// SIMATIC S7-200 project (STEP 7-Micro/WIN), CPU 224XP REL 02.01

SYMBOL_TABLE USUARIO1
S_LENTO          I0.0
S_RAPIDO         I0.1
B_LENTO          I0.2
B_RAPIDO         I0.3
D_LENTO          I0.4
D_RAPIDO         I0.5
I_LENTO          I0.6
I_RAPIDO         I0.7
FC_BAJADA        I1.0
FC_SUBIDA        I1.1
FC_IZQUIERDA     I1.2
FC_DERECHA       I1.3
M1_S_U1V1W1TSR   Q0.0
M1_S_U2V2W2_TSR  Q0.1
M1_SB_CORTOCIRQUITADO Q0.2
M1_B_U1V1W1_RST  Q0.3
M1_B_U2V2W2_RST  Q0.4
M2_D_U1V1W1_RST  Q0.5
M2_D_U2V2W2_RST  Q0.6
M2_DI_CORTOCIRQUITADO Q0.7
M2_I_U1V1W1_TSR  Q1.0
M2_I_U2V2W2_TSR  Q1.1
END_SYMBOL_TABLE

ORGANIZATION_BLOCK PRINCIPAL:OB1
TITLE=COMENTARIOS DEL PROGRAMA
BEGIN
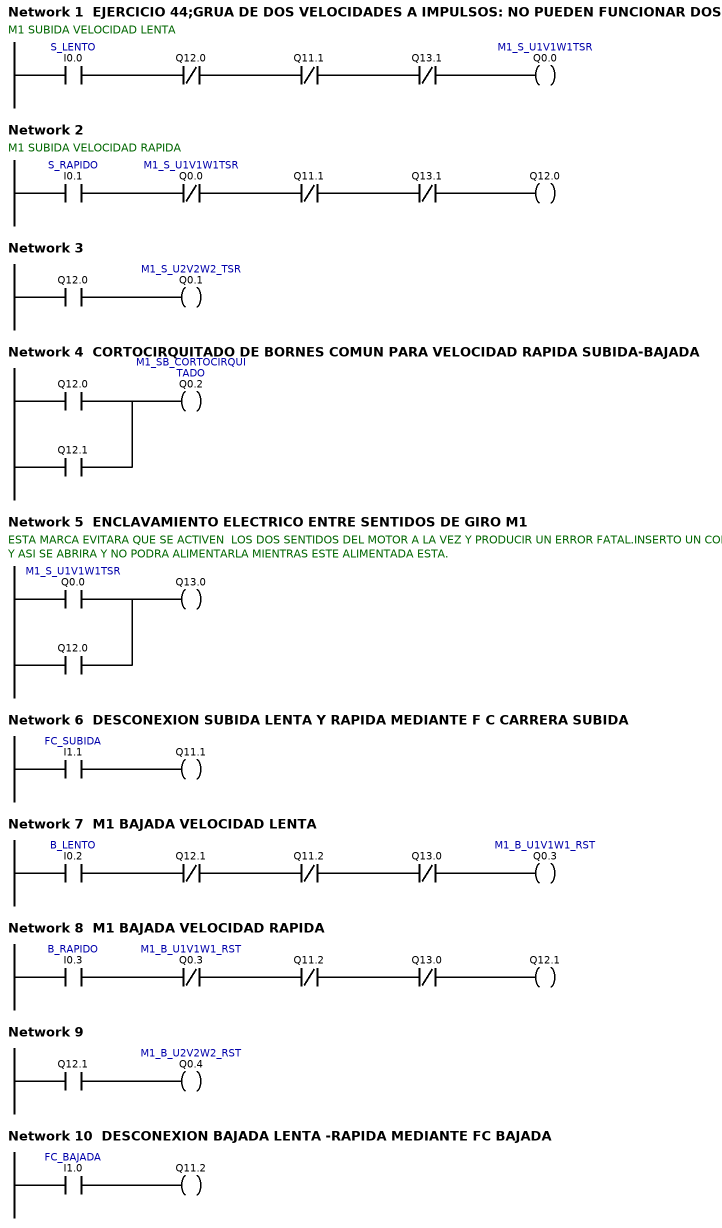
Network 1 // EJERCICIO 44;GRUA DE DOS VELOCIDADES A IMPULSOS:
NO PUEDEN FUNCIONAR DOS VELOCIDADES DEL MISMO SENTIDO A LA VEZ Y TAMPOCO DOS SENTIDOS DEL MISMO MOTOR.
// M1 SUBIDA VELOCIDAD LENTA
LD     S_LENTO:I0.0
AN     Q12.0
AN     Q11.1
AN     Q13.1
=      M1_S_U1V1W1TSR:Q0.0
Network 2
// M1 SUBIDA VELOCIDAD RAPIDA
LD     S_RAPIDO:I0.1
AN     M1_S_U1V1W1TSR:Q0.0
AN     Q11.1
AN     Q13.1
=      Q12.0
Network 3
LD     Q12.0
=      M1_S_U2V2W2_TSR:Q0.1
Network 4 // CORTOCIRQUITADO DE BORNES COMUN PARA VELOCIDAD RAPIDA SUBIDA-BAJADA
LD     Q12.0
O      Q12.1
=      M1_SB_CORTOCIRQUITADO:Q0.2
Network 5 // ENCLAVAMIENTO ELECTRICO ENTRE SENTIDOS DE GIRO M1
// ESTA MARCA EVITARA QUE SE ACTIVEN  LOS DOS SENTIDOS DEL MOTOR A LA VEZ Y PRODUCIR UN ERROR FATAL.INSERTO UN CONTACTO CERRADO DELANTE DE LA BOBINA DEL SENTIDO CONTRARIO Y ASI SE ABRIRA Y NO PODRA ALIMENTARLA MIENTRAS ESTE ALIMENTADA ESTA.
LD     M1_S_U1V1W1TSR:Q0.0
O      Q12.0
=      Q13.0
Network 6 // DESCONEXION SUBIDA LENTA Y RAPIDA MEDIANTE F C CARRERA SUBIDA
LD     FC_SUBIDA:I1.1
=      Q11.1
Network 7 // M1 BAJADA VELOCIDAD LENTA 
LD     B_LENTO:I0.2
AN     Q12.1
AN     Q11.2
AN     Q13.0
=      M1_B_U1V1W1_RST:Q0.3
Network 8 // M1 BAJADA VELOCIDAD RAPIDA
LD     B_RAPIDO:I0.3
AN     M1_B_U1V1W1_RST:Q0.3
AN     Q11.2
AN     Q13.0
=      Q12.1
Network 9
LD     Q12.1
=      M1_B_U2V2W2_RST:Q0.4
Network 10 // DESCONEXION BAJADA LENTA -RAPIDA MEDIANTE FC BAJADA
LD     FC_BAJADA:I1.0
=      Q11.2
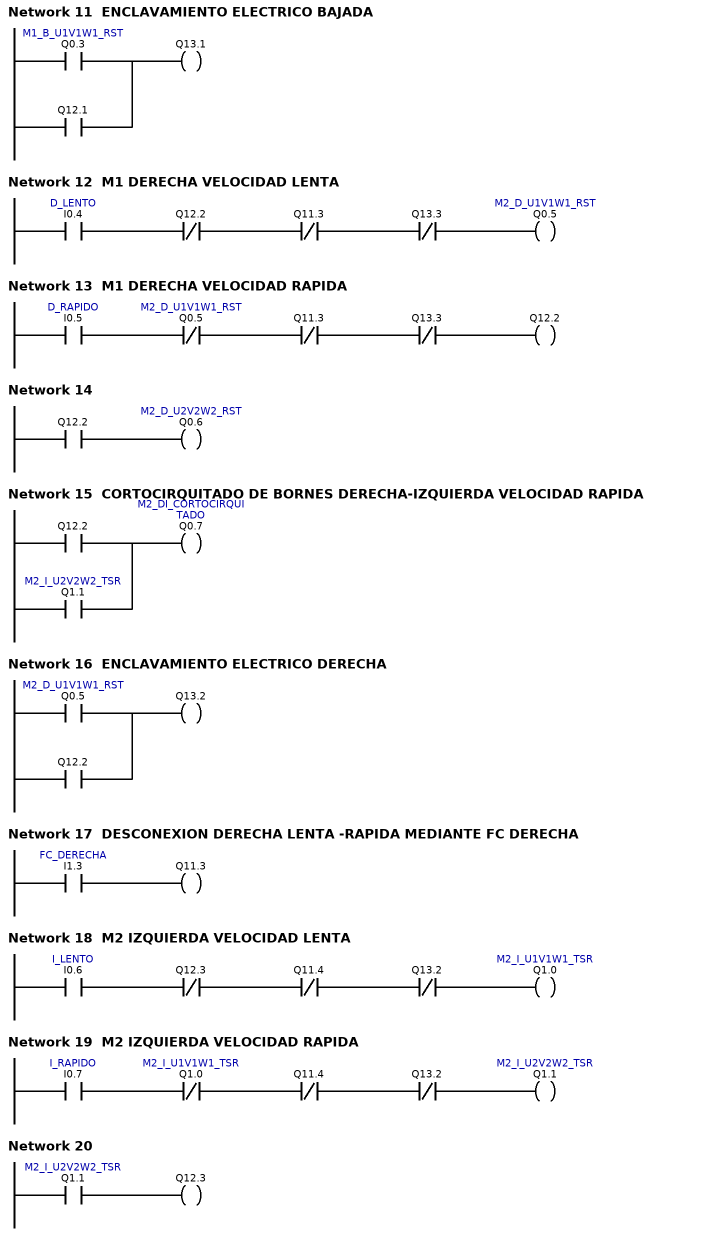
Network 11 // ENCLAVAMIENTO ELECTRICO BAJADA
LD     M1_B_U1V1W1_RST:Q0.3
O      Q12.1
=      Q13.1
Network 12 // M1 DERECHA VELOCIDAD LENTA 
LD     D_LENTO:I0.4
AN     Q12.2
AN     Q11.3
AN     Q13.3
=      M2_D_U1V1W1_RST:Q0.5
Network 13 // M1 DERECHA VELOCIDAD RAPIDA
LD     D_RAPIDO:I0.5
AN     M2_D_U1V1W1_RST:Q0.5
AN     Q11.3
AN     Q13.3
=      Q12.2
Network 14
LD     Q12.2
=      M2_D_U2V2W2_RST:Q0.6
Network 15 // CORTOCIRQUITADO DE BORNES DERECHA-IZQUIERDA VELOCIDAD RAPIDA
LD     Q12.2
O      M2_I_U2V2W2_TSR:Q1.1
=      M2_DI_CORTOCIRQUITADO:Q0.7
Network 16 // ENCLAVAMIENTO ELECTRICO DERECHA
LD     M2_D_U1V1W1_RST:Q0.5
O      Q12.2
=      Q13.2
Network 17 // DESCONEXION DERECHA LENTA -RAPIDA MEDIANTE FC DERECHA
LD     FC_DERECHA:I1.3
=      Q11.3
Network 18 // M2 IZQUIERDA VELOCIDAD LENTA 
LD     I_LENTO:I0.6
AN     Q12.3
AN     Q11.4
AN     Q13.2
=      M2_I_U1V1W1_TSR:Q1.0
Network 19 // M2 IZQUIERDA VELOCIDAD RAPIDA
LD     I_RAPIDO:I0.7
AN     M2_I_U1V1W1_TSR:Q1.0
AN     Q11.4
AN     Q13.2
=      M2_I_U2V2W2_TSR:Q1.1
Network 20
LD     M2_I_U2V2W2_TSR:Q1.1
=      Q12.3
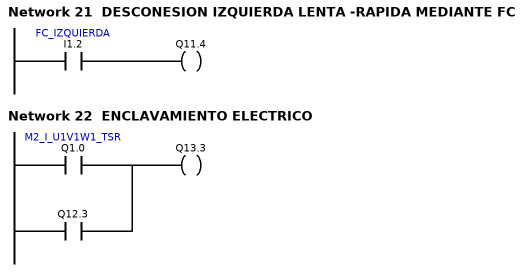
Network 21 // DESCONESION IZQUIERDA LENTA -RAPIDA MEDIANTE FC IZQUIERDA
LD     FC_IZQUIERDA:I1.2
=      Q11.4
Network 22 // ENCLAVAMIENTO ELECTRICO
LD     M2_I_U1V1W1_TSR:Q1.0
O      Q12.3
=      Q13.3
END_ORGANIZATION_BLOCK
